{attribute 'qualified_only'}
VAR_GLOBAL
END_VAR

(* stored: Version 1.1.0.1, ProductVersion 3.1.4022.7
   GVL GVL_05_Manual_Servo_Motor_Shelf_Y: Id {00917c76-9139-41ea-93a7-e95f28e695e8} *)
